// Returns Unix-relative system time in 100 ns ticks.
FUNCTION GetUnixTime : ULINT
VAR_INPUT
	nOffset : LINT := 0; // Offset applied before epoch conversion.
END_VAR
VAR
END_VAR

GetUnixTime := Tc2_System.F_GetSystemTime() - LINT_TO_ULINT(11_644_473_678_000_000_0 + nOffset);

END_FUNCTION

(* stored: Version 1.1.0.1
   POU GetUnixTime: Id {2743d7a2-b5ef-4e7a-a5e4-a656ba43ea9a}, SpecialFunc None *)
